TYPE Taak_1 :
	(
		NieuweOrderGaragist,
		VoorraadAdministratief,
		VerzamelingArtikelen,
		OrderGeanuleerd
	) := NieuweOrderGaragist;
END_TYPE

(* stored: Version 1.1.0.1, ProductVersion 3.1.4024.12
   DUT Taak_1: Id {4dc2f315-6e55-411e-b7c1-780b357820cb} *)
